PROGRAM MAIN
VAR
END_VAR

END_PROGRAM

(* stored: Version 1.1.0.1
   POU MAIN: Id {a546692e-f77d-4dc9-b456-635ae84187da} *)
